// TIA Portal V20 export
DATA_BLOCK "DB_Part_Data"   // DB131
// stored: InstanceOfName FB_Part_Data, InstanceOfType FB
"FB_Part_Data"
   // VAR
   //    Part_Data_Ident : "FB_ReadWrite_GUDs";
   //    sWriteDataEnable { S7_SetPoint := 'True'} : Bool;
   //    sNewPartDataIdent : Bool;
   //    RT_NewPartDataIdent : R_TRIG;
   //    sCurrentPartDataIdent { S7_SetPoint := 'True'} : String;
   // END_VAR
BEGIN
END_DATA_BLOCK
